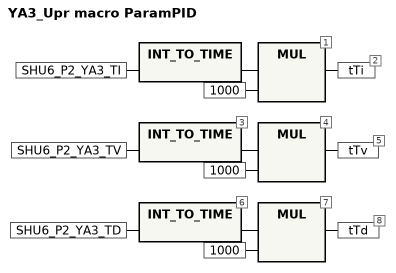
[picture p362: YA3_Upr macro ParamPID (CFC)]
_CFC_ (* Continuous Function Chart, elements in execution order *)
#0 TON_SHU6_P2_P1_DI7_RUN:TON(IN: SHU6_P2_P1_DI7_RUN, PT: T#10s)
#1 AND(NOT SHU6_P2_UST_RE_RABOTA, #0.Q, NOT SHU6_P2_UST_RE_PROGREV)
#2 reg2 <= #1
#3 AND(SHU6_P2_UST_RE_RABOTA, #0.Q)
#4 reg1 <= #3
#5 AND(reg1, SHU6_P2_TE6_T_DOST)
#6 AND(reg2, SHU6_P2_TE4_DOST)
#7 OR(#5, #6)
#8 YA3_DOST <= #7
#9 MACRO ParamPID()
	#10 INT_TO_TIME(SHU6_P2_YA3_TI)
	#11 MUL(#10, 1000)
	#12 tTi <= #11
	#13 INT_TO_TIME(SHU6_P2_YA3_TV)
	#14 MUL(#13, 1000)
	#15 tTv <= #14
	#16 INT_TO_TIME(SHU6_P2_YA3_TD)
	#17 MUL(#16, 1000)
	#18 tTd <= #17
END_MACRO
#19 SUB(SHU6_P2_TE6_T_UST, SHU6_P2_TE4_VN)
#20 EPS2 <= #19
#21 SUB(SHU6_P2_TE6_T_UST, SHU6_P2_TE6_T_VN)
#22 EPS1 <= #21
#23 SEL(reg1, SHU6_P2_TE4_UST, SHU6_P2_TE6_T_UST)
#24 >(EPS1, EPS2)
#25 AND(reg1, #24)
#26 SEL(#25, SHU6_P2_TE4_VN, SHU6_P2_TE6_T_VN)
#27 OR(reg1, reg2)
#28 AND(#27, YA3_DOST)
#29 SEL(#28, 0, #23)
#30 SEL(#28, 0, #26)
#31 AND(#28, SHU6_P2_YA3_SA4_DI1_A)
#32 SHU6_P2_YA3_AUTO <= #31
#33 AND(NOT SHU6_P2_TE1_B_UST_MYAG_REG, SHU6_P2_UST_RE_PROGREV)
#34 OR(Z_ZAM_SR, #33)
#35 AND(#31, NOT #34)
#36 AND(#35, NOT SHU6_P2_Z_GVS1_OTKAZ)
#37 YA3_REG_POL <= #36
#38 SEL(#36, eHVACCtrlMode_Manual, eHVACCtrlMode_Auto)
#39 SEL(NOT SHU6_P2_P1_DI7_RUN, SHU6_P2_YA3_UP_VN, rYMin)
#40 SEL(SHU6_P2_UST_RE_PROGREV, #39, 50)
#41 SEL(#34, #40, 100)
#42 SEL(SHU6_P2_YA3_SA4_DI1_A, SHU6_P2_YA3_UP_VN, #41)
#43 SEL(SHU6_P2_Z_GVS1_OTKAZ, #42, 0)
#44 YA3_PID:FB_HVACPIDCtrl(eHVACDataSecurityType_Idle, FALSE, TRUE, #29, #30, tTaskCycleTime, tTaskCycleTime, #38, #43, SHU6_P2_YA3_UP_VN, FALSE, SHU6_P2_SB, deadRange, direction, SHU6_P2_YA3_KP, tTi, tTv, tTd, rYMin, rYMax)
#45 SHU6_P2_YA3_RASSOG <= #44.out 2
#46 YA3_OTKAZ <= #44.out 8
#47 SEL(SHU6_P2_YA3_SA4_DI1_A, 0, #44.out 1)
#48 SHU6_P2_YA3_ZAD_VN <= #47
#49 SUB(#47, SHU6_P2_YA3_UP_VN)
#50 SHU6_P2_YA3_RASSOG_POL <= #49
#51 SEL(SHU6_P2_UST_ZIMA, 0, SHU6_P2_YA3_UP_MIN)
#52 rYMin <= #51
_END_CFC_
END_PROGRAM

(* POU IM/YA4_Upr, CFC *)
PROGRAM YA4_Upr
VAR
	YA4_PID: FB_HVACPIDCtrl;

	deadRange: REAL := 0.1;
	direction: BOOL := TRUE;
	tTi: TIME;
	tTv: TIME;
	tTd: TIME;

	rYMin: REAL := 0;
	rYMax: REAL := 100;
	YA4_OTAZ: BOOL;
END_VAR
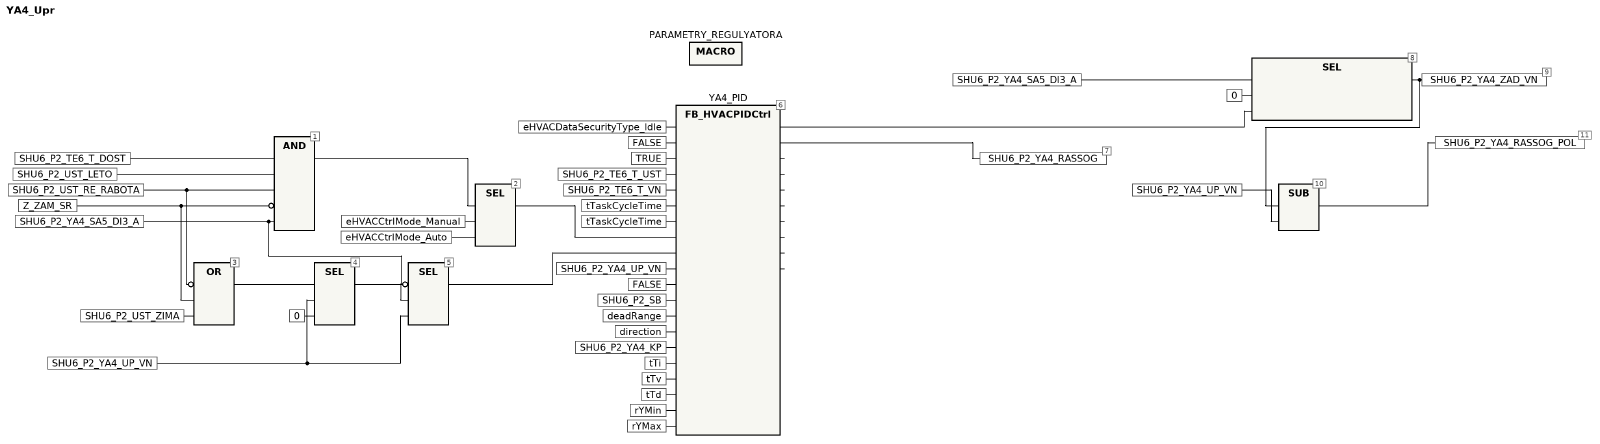
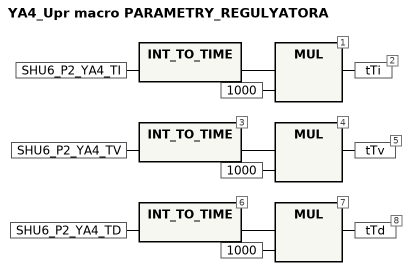
_CFC_ (* Continuous Function Chart, elements in execution order *)
#0 MACRO PARAMETRY_REGULYATORA()
	#1 INT_TO_TIME(SHU6_P2_YA4_TI)
	#2 MUL(#1, 1000)
	#3 tTi <= #2
	#4 INT_TO_TIME(SHU6_P2_YA4_TV)
	#5 MUL(#4, 1000)
	#6 tTv <= #5
	#7 INT_TO_TIME(SHU6_P2_YA4_TD)
	#8 MUL(#7, 1000)
	#9 tTd <= #8
END_MACRO
#10 AND(SHU6_P2_TE6_T_DOST, SHU6_P2_UST_LETO, SHU6_P2_UST_RE_RABOTA, NOT Z_ZAM_SR, SHU6_P2_YA4_SA5_DI3_A)
#11 SEL(#10, eHVACCtrlMode_Manual, eHVACCtrlMode_Auto)
#12 OR(NOT SHU6_P2_UST_RE_RABOTA, Z_ZAM_SR, SHU6_P2_UST_ZIMA)
#13 SEL(#12, SHU6_P2_YA4_UP_VN, 0)
#14 SEL(NOT SHU6_P2_YA4_SA5_DI3_A, #13, SHU6_P2_YA4_UP_VN)
#15 YA4_PID:FB_HVACPIDCtrl(eHVACDataSecurityType_Idle, FALSE, TRUE, SHU6_P2_TE6_T_UST, SHU6_P2_TE6_T_VN, tTaskCycleTime, tTaskCycleTime, #11, #14, SHU6_P2_YA4_UP_VN, FALSE, SHU6_P2_SB, deadRange, direction, SHU6_P2_YA4_KP, tTi, tTv, tTd, rYMin, rYMax)
#16 SHU6_P2_YA4_RASSOG <= #15.out 2
#17 SEL(SHU6_P2_YA4_SA5_DI3_A, 0, #15.out 1)
#18 SHU6_P2_YA4_ZAD_VN <= #17
#19 SUB(#17, SHU6_P2_YA4_UP_VN)
#20 SHU6_P2_YA4_RASSOG_POL <= #19
_END_CFC_
END_PROGRAM

(* POU Output/ALL_Output, CFC *)
PROGRAM ALL_Output
VAR
END_VAR
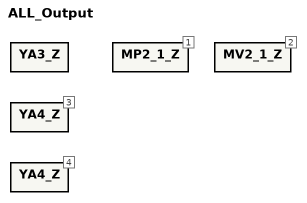
_CFC_ (* Continuous Function Chart, elements in execution order *)
#0 YA3_Z()
#1 MP2_1_Z()
#2 MV2_1_Z()
#3 YA4_Z()
#4 YA4_Z()
_END_CFC_
(* the same logic as Structured Text *)
YA3_Z();
MP2_1_Z();
MV2_1_Z();
YA4_Z();
YA4_Z();
END_PROGRAM

(* POU Output/AO/YA3_Z, CFC *)
PROGRAM YA3_Z
VAR
	fb_HVACAO_SHU6_P2_YA3_AO7: FB_HVACAnalogOutput;
	enableFeedbCtrl: BOOL := FALSE;
	hysFbCtrl: REAL := 0;
	direction: BOOL;
	delay: TIME := T#0s;
END_VAR
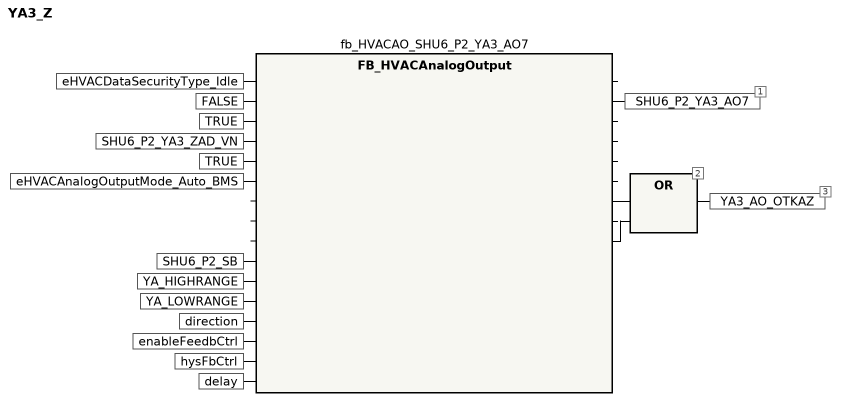
_CFC_ (* Continuous Function Chart, elements in execution order *)
#0 fb_HVACAO_SHU6_P2_YA3_AO7:FB_HVACAnalogOutput(eHVACDataSecurityType_Idle, FALSE, TRUE, SHU6_P2_YA3_ZAD_VN, TRUE, eHVACAnalogOutputMode_Auto_BMS, -, -, -, SHU6_P2_SB, YA_HIGHRANGE, YA_LOWRANGE, direction, enableFeedbCtrl, hysFbCtrl, delay)
#1 SHU6_P2_YA3_AO7 <= #0.out 2
#2 OR(#0.out 7, #0.out 9)
#3 YA3_AO_OTKAZ <= #2
_END_CFC_
END_PROGRAM

(* POU Output/AO/MP2_1_Z, CFC *)
PROGRAM MP2_1_Z
VAR
	fb_HVACAO_SHU6_P2_UZ1_1_AO1: FB_HVACAnalogOutput;
	enableFeedbCtrl: BOOL := FALSE;
	hysFbCtrl: REAL := 0;
	direction: BOOL;
	delay: TIME := T#0s;
	hi: REAL := 50;
	low: REAL := 0;

END_VAR
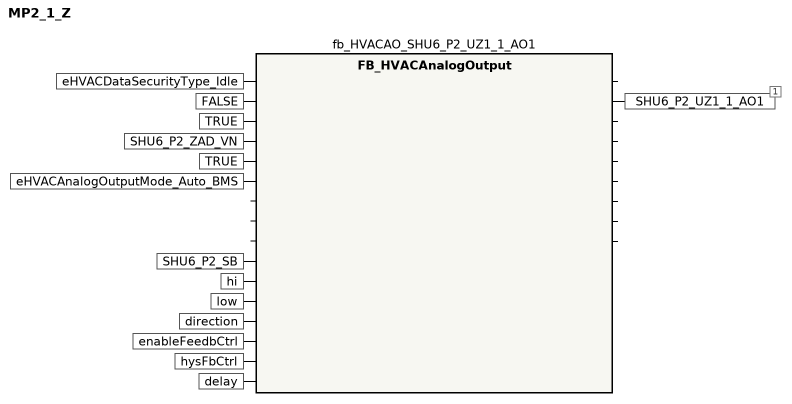
_CFC_ (* Continuous Function Chart, elements in execution order *)
#0 fb_HVACAO_SHU6_P2_UZ1_1_AO1:FB_HVACAnalogOutput(eHVACDataSecurityType_Idle, FALSE, TRUE, SHU6_P2_ZAD_VN, TRUE, eHVACAnalogOutputMode_Auto_BMS, -, -, -, SHU6_P2_SB, hi, low, direction, enableFeedbCtrl, hysFbCtrl, delay)
#1 SHU6_P2_UZ1_1_AO1 <= #0.out 2
_END_CFC_
END_PROGRAM

(* POU Output/AO/MV2_1_Z, CFC *)
PROGRAM MV2_1_Z
VAR
	fb_HVACAO_SHU6_V2_UZ2_1_AO3: FB_HVACAnalogOutput;
	enableFeedbCtrl: BOOL := FALSE;
	hysFbCtrl: REAL := 0;
	direction: BOOL;
	delay: TIME := T#0s;
	hi: REAL := 50;
	low: REAL := 0;


END_VAR
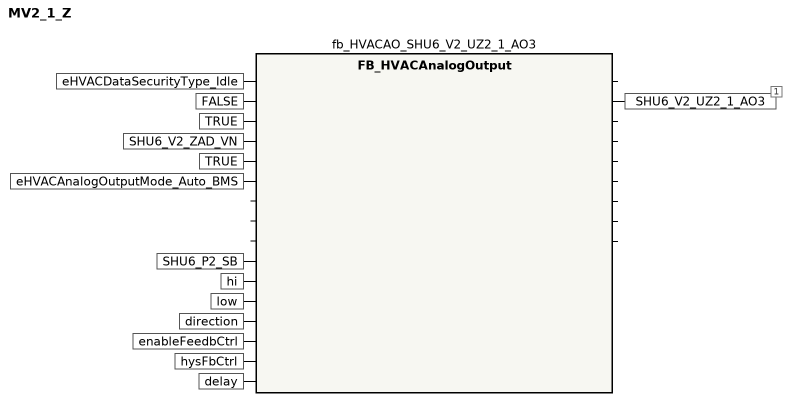
_CFC_ (* Continuous Function Chart, elements in execution order *)
#0 fb_HVACAO_SHU6_V2_UZ2_1_AO3:FB_HVACAnalogOutput(eHVACDataSecurityType_Idle, FALSE, TRUE, SHU6_V2_ZAD_VN, TRUE, eHVACAnalogOutputMode_Auto_BMS, -, -, -, SHU6_P2_SB, hi, low, direction, enableFeedbCtrl, hysFbCtrl, delay)
#1 SHU6_V2_UZ2_1_AO3 <= #0.out 2
_END_CFC_
END_PROGRAM

(* POU Output/AO/YA4_Z, CFC *)
PROGRAM YA4_Z
VAR
	fb_HVACAO_SHU6_P2_YA4_AO1: FB_HVACAnalogOutput;
	enableFeedbCtrl: BOOL := FALSE;
	hysFbCtrl: REAL := 0;
	direction: BOOL;
	delay: TIME := T#0s;
END_VAR
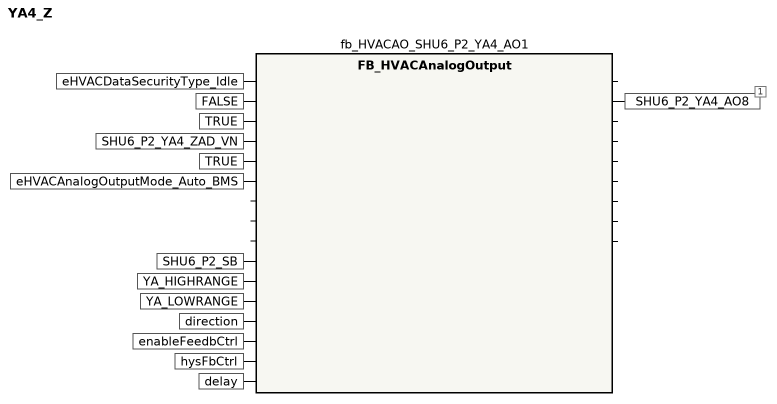
_CFC_ (* Continuous Function Chart, elements in execution order *)
#0 fb_HVACAO_SHU6_P2_YA4_AO1:FB_HVACAnalogOutput(eHVACDataSecurityType_Idle, FALSE, TRUE, SHU6_P2_YA4_ZAD_VN, TRUE, eHVACAnalogOutputMode_Auto_BMS, -, -, -, SHU6_P2_SB, YA_HIGHRANGE, YA_LOWRANGE, direction, enableFeedbCtrl, hysFbCtrl, delay)
#1 SHU6_P2_YA4_AO8 <= #0.out 2
_END_CFC_
END_PROGRAM

(* POU Input/CI/ModBus_M, CFC *)
PROGRAM ModBus_M
VAR
	MB_READ_REGS: ModbusRtuMaster_KL6x22B;
	Quantity: WORD:= 1;
	MBAddr: WORD:= 16#3000;
	MBAddr_1: WORD:= 16#0C82;
	CTU_ModBus: CTU;
	TON1: TON;
	TON2: TON;


	RT_ModBus: R_TRIG;

	Errorld: MODBUS_ERRORS;
	cbRead: UINT;
END_VAR
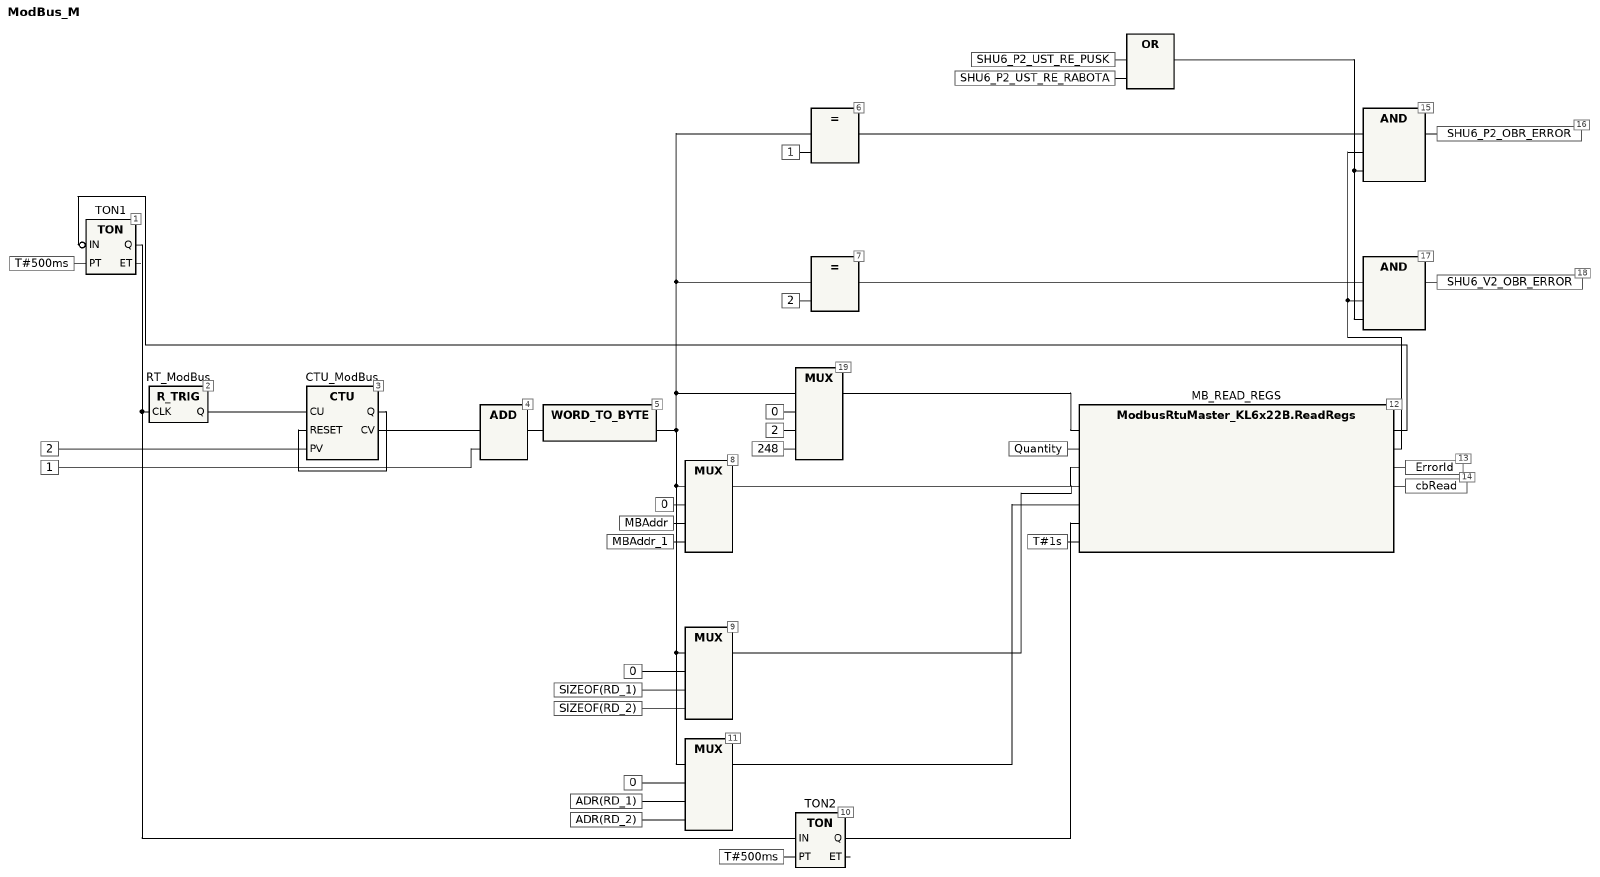
